Staubli VAL3: OnEvent4.pgx

program OnEvent4()
begin
  //-----------------------------------------------------------------------
  //Header begin
  //LasMAN3.7
  //Description of program
  //
  //Input parameters
  //
  //Output paramaters
  //Example
  //  call OnEvent1()
  //History
  //  Creation : 2013-06-23  y.ye@staubli.com
  //Header end
  //-----------------------------------------------------------------------

  call Teach:TeachAction()
  DataBase:nInterfaceType=9
end
